{attribute addProperty BoxType "EJ5002-0000-0016"}
{attribute addProperty Id "SSI_Inputs_ChannelAT %I*ARRAY[0..1] OF SSI_Inputs_Channel_F7D238D196120WcStateAT %I*WcState_F855686C1620InfoDataAT %I*InfoData_BC63D37F80100"}
{attribute addProperty CRC "2301877599"}
{attribute addProperty SizeInBites "192"}
{attribute addProperty SizeInBytes "24"}
TYPE EJ5002_8CF434FD :
STRUCT
	{attribute addProperty Name "SSI_Inputs_Channel"}
	SSI_Inputs_Channel : ARRAY[0..1] OF SSI_Inputs_Channel_F7D238D1;
	{attribute addProperty Name "WcState"}
	WcState : WcState_F855686C;
	{attribute addProperty Name "InfoData"}
	InfoData : InfoData_BC63D37F;
END_STRUCT
END_TYPE

(* stored: Version 1.2.0.0, ProductVersion 3.1.4024.9
   DUT EJ5002_8CF434FD: Id {9038b48a-ed8f-4d18-9f08-1067fbae8ff9} *)
